FUNCTION_BLOCK FB_Timer
VAR_INPUT
	bEnable 	: BOOL;
	bStart 		: BOOL;
	bStop 		: BOOL;
	fCycleTime  : LREAL;
END_VAR
VAR_OUTPUT
	fTime : LREAL;
END_VAR
VAR
END_VAR

IF bStart AND NOT(bStop) AND bEnable THEN
	fTime := fTime + fCycleTime;
ELSE
	fTime := 0.0;
END_IF

END_FUNCTION_BLOCK

(* stored: Version 1.1.0.1, ProductVersion 3.1.4024.12
   POU FB_Timer: Id {5e9d1a3a-15af-4ea9-89ef-71fde47ab25e}, SpecialFunc None *)
